(* PLC project Logging example, Unknown Generic PLC 1 *)
(* stored: creationDateTime 2013-01-29T14:01:00, contentDescription This example shows logging functionality in Beremiz. Here are shown two ways of logging: - from IEC PLC program; - from python extension., modificationDateTime 2025-05-13T10:52:05 *)

FUNCTION_BLOCK C_Pragma
  VAR_INPUT
    TRIG : BOOL;
    IN : INT;
  END_VAR
  VAR
    rtrig : R_TRIG;
  END_VAR

            rtrig(CLK := TRIG);
IF rtrig.Q THEN 
{{
  short inval = GetFbVar(IN);
  printf("C runtime OK #%d\n", inval);
  fflush(stdout);
}}
END_IF;

          
END_FUNCTION_BLOCK

PROGRAM program0
  VAR
    beat : BOOL;
    count : INT;
    LOGGER0 : LOGGER;
    lvl : LOGLEVEL := INFO;
    Timer : TOF;
    C_Pragma0 : C_Pragma;
    EXIT_SIM0 : EXIT_SIM;
    SIM_PRINT0 : SIM_PRINT;
  END_VAR
  VAR  (* added by the conversion: wires and edge detectors of the diagram *)
    _NOT3_OUT : BOOL;
    R_TRIG1 : R_TRIG;
    _ADD5_OUT : INT;
    _CONCAT8_OUT : STRING;
  END_VAR

(* FBD diagram, written out as Structured Text *)
Timer(IN := beat, PT := T#1s);
_NOT3_OUT := NOT Timer.Q;
beat := _NOT3_OUT;
R_TRIG1(CLK := _NOT3_OUT);
_ADD5_OUT := BOOL_TO_INT(R_TRIG1.Q) + count;
count := _ADD5_OUT;
_CONCAT8_OUT := CONCAT('C runtime log OK #', INT_TO_STRING(_ADD5_OUT));
LOGGER0(TRIG := _NOT3_OUT, MSG := _CONCAT8_OUT, LEVEL := lvl);
C_Pragma0(TRIG := _NOT3_OUT, IN := _ADD5_OUT);
EXIT_SIM0(TRIG := _ADD5_OUT > 10, EXIT_CODE := 42);
SIM_PRINT0(TRIG := _NOT3_OUT, MSG := _CONCAT8_OUT);
END_PROGRAM

CONFIGURATION config
  RESOURCE resource1 ON PLC
    TASK task0(INTERVAL := T#100ms, PRIORITY := 0);
    PROGRAM prg WITH task0 : program0;
  END_RESOURCE
END_CONFIGURATION
